def cycle_3():
  # --- Cycle 3 - Circulaire (UI) ---
  movel(apply_correction(p[-0.017788, 0.586142, 0.060004, 3.141576, 0.000000, 0.000000]), a=URSCRIPT_ACCEL*ACCEL_FACTOR, v=0.2500*SPEED_FACTOR)
  sleep(0.2)
  zero_ftsensor()
  sleep(0.2)
  force_mode(MEAS_FRAME, [0, 0, 1, 0, 0, 0], [0, 0, -6.0, 0, 0, 0], 2, [0.008, 0.008, 0.04, 0.35, 0.35, 0.35])
  movel(apply_correction(p[-0.017788, 0.586142, 0.045004, 3.141576, 0.000000, 0.000000]), a=URSCRIPT_ACCEL*ACCEL_FACTOR, v=URSCRIPT_RECONTACT_V*SPEED_FACTOR)
  movel(apply_correction(p[-0.017788, 0.586142, 0.050004, 3.141576, 0.000000, 0.000000]), a=URSCRIPT_ACCEL*ACCEL_FACTOR, v=V_CIRC*SPEED_FACTOR, r=URSCRIPT_BLEND)
  movel(apply_correction(p[-0.011098, 0.583533, 0.050004, 3.141576, 0.000000, 0.000000]), a=URSCRIPT_ACCEL*ACCEL_FACTOR, v=V_CIRC*SPEED_FACTOR, r=URSCRIPT_BLEND)
  movel(apply_correction(p[-0.004916, 0.587048, 0.050004, 3.141576, 0.000000, 0.000000]), a=URSCRIPT_ACCEL*ACCEL_FACTOR, v=V_CIRC*SPEED_FACTOR, r=URSCRIPT_BLEND)
  movel(apply_correction(p[-0.005086, 0.594004, 0.050004, 3.141576, 0.000000, 0.000000]), a=URSCRIPT_ACCEL*ACCEL_FACTOR, v=V_CIRC*SPEED_FACTOR, r=URSCRIPT_BLEND)
  movel(apply_correction(p[-0.011712, 0.596025, 0.050004, 3.141576, 0.000000, 0.000000]), a=URSCRIPT_ACCEL*ACCEL_FACTOR, v=V_CIRC*SPEED_FACTOR, r=URSCRIPT_BLEND)
  movel(apply_correction(p[-0.016472, 0.590781, 0.050004, 3.141576, 0.000000, 0.000000]), a=URSCRIPT_ACCEL*ACCEL_FACTOR, v=V_CIRC*SPEED_FACTOR, r=URSCRIPT_BLEND)
  movel(apply_correction(p[-0.015164, 0.583730, 0.050004, 3.141576, 0.000000, 0.000000]), a=URSCRIPT_ACCEL*ACCEL_FACTOR, v=V_CIRC*SPEED_FACTOR, r=URSCRIPT_BLEND)
  movel(apply_correction(p[-0.009065, 0.579930, 0.050004, 3.141576, 0.000000, 0.000000]), a=URSCRIPT_ACCEL*ACCEL_FACTOR, v=V_CIRC*SPEED_FACTOR, r=URSCRIPT_BLEND)
  movel(apply_correction(p[-0.002264, 0.582086, 0.050004, 3.141576, 0.000000, 0.000000]), a=URSCRIPT_ACCEL*ACCEL_FACTOR, v=V_CIRC*SPEED_FACTOR, r=URSCRIPT_BLEND)
  movel(apply_correction(p[-0.000623, 0.588885, 0.050004, 3.141576, 0.000000, 0.000000]), a=URSCRIPT_ACCEL*ACCEL_FACTOR, v=V_CIRC*SPEED_FACTOR, r=URSCRIPT_BLEND)
  movel(apply_correction(p[-0.006418, 0.592643, 0.050004, 3.141576, 0.000000, 0.000000]), a=URSCRIPT_ACCEL*ACCEL_FACTOR, v=V_CIRC*SPEED_FACTOR, r=URSCRIPT_BLEND)
  movel(apply_correction(p[-0.012226, 0.588648, 0.050004, 3.141576, 0.000000, 0.000000]), a=URSCRIPT_ACCEL*ACCEL_FACTOR, v=V_CIRC*SPEED_FACTOR, r=URSCRIPT_BLEND)
  movel(apply_correction(p[-0.012291, 0.581489, 0.050004, 3.141576, 0.000000, 0.000000]), a=URSCRIPT_ACCEL*ACCEL_FACTOR, v=V_CIRC*SPEED_FACTOR, r=URSCRIPT_BLEND)
  movel(apply_correction(p[-0.006988, 0.576638, 0.050004, 3.141576, 0.000000, 0.000000]), a=URSCRIPT_ACCEL*ACCEL_FACTOR, v=V_CIRC*SPEED_FACTOR, r=URSCRIPT_BLEND)
  movel(apply_correction(p[0.000125, 0.577386, 0.050004, 3.141576, 0.000000, 0.000000]), a=URSCRIPT_ACCEL*ACCEL_FACTOR, v=V_CIRC*SPEED_FACTOR, r=URSCRIPT_BLEND)
  movel(apply_correction(p[0.003408, 0.583603, 0.050004, 3.141576, 0.000000, 0.000000]), a=URSCRIPT_ACCEL*ACCEL_FACTOR, v=V_CIRC*SPEED_FACTOR, r=URSCRIPT_BLEND)
  movel(apply_correction(p[-0.001104, 0.588825, 0.050004, 3.141576, 0.000000, 0.000000]), a=URSCRIPT_ACCEL*ACCEL_FACTOR, v=V_CIRC*SPEED_FACTOR, r=URSCRIPT_BLEND)
  movel(apply_correction(p[-0.007670, 0.586361, 0.050004, 3.141576, 0.000000, 0.000000]), a=URSCRIPT_ACCEL*ACCEL_FACTOR, v=V_CIRC*SPEED_FACTOR, r=URSCRIPT_BLEND)
  movel(apply_correction(p[-0.009144, 0.579371, 0.050004, 3.141576, 0.000000, 0.000000]), a=URSCRIPT_ACCEL*ACCEL_FACTOR, v=V_CIRC*SPEED_FACTOR, r=URSCRIPT_BLEND)
  movel(apply_correction(p[-0.004813, 0.573634, 0.050004, 3.141576, 0.000000, 0.000000]), a=URSCRIPT_ACCEL*ACCEL_FACTOR, v=V_CIRC*SPEED_FACTOR, r=URSCRIPT_BLEND)
  movel(apply_correction(p[0.002324, 0.572985, 0.050004, 3.141576, 0.000000, 0.000000]), a=URSCRIPT_ACCEL*ACCEL_FACTOR, v=V_CIRC*SPEED_FACTOR, r=URSCRIPT_BLEND)
  movel(apply_correction(p[0.006999, 0.578286, 0.050004, 3.141576, 0.000000, 0.000000]), a=URSCRIPT_ACCEL*ACCEL_FACTOR, v=V_CIRC*SPEED_FACTOR, r=URSCRIPT_BLEND)
  movel(apply_correction(p[0.004110, 0.584567, 0.050004, 3.141576, 0.000000, 0.000000]), a=URSCRIPT_ACCEL*ACCEL_FACTOR, v=V_CIRC*SPEED_FACTOR, r=URSCRIPT_BLEND)
  movel(apply_correction(p[-0.002829, 0.583846, 0.050004, 3.141576, 0.000000, 0.000000]), a=URSCRIPT_ACCEL*ACCEL_FACTOR, v=V_CIRC*SPEED_FACTOR, r=URSCRIPT_BLEND)
  movel(apply_correction(p[-0.005691, 0.577324, 0.050004, 3.141576, 0.000000, 0.000000]), a=URSCRIPT_ACCEL*ACCEL_FACTOR, v=V_CIRC*SPEED_FACTOR, r=URSCRIPT_BLEND)
  movel(apply_correction(p[-0.002490, 0.570894, 0.050004, 3.141576, 0.000000, 0.000000]), a=URSCRIPT_ACCEL*ACCEL_FACTOR, v=V_CIRC*SPEED_FACTOR, r=URSCRIPT_BLEND)
  movel(apply_correction(p[0.004406, 0.568905, 0.050004, 3.141576, 0.000000, 0.000000]), a=URSCRIPT_ACCEL*ACCEL_FACTOR, v=V_CIRC*SPEED_FACTOR, r=URSCRIPT_BLEND)
  movel(apply_correction(p[0.010171, 0.573044, 0.050004, 3.141576, 0.000000, 0.000000]), a=URSCRIPT_ACCEL*ACCEL_FACTOR, v=V_CIRC*SPEED_FACTOR, r=URSCRIPT_BLEND)
  movel(apply_correction(p[0.009098, 0.579900, 0.050004, 3.141576, 0.000000, 0.000000]), a=URSCRIPT_ACCEL*ACCEL_FACTOR, v=V_CIRC*SPEED_FACTOR, r=URSCRIPT_BLEND)
  movel(apply_correction(p[0.002251, 0.581029, 0.050004, 3.141576, 0.000000, 0.000000]), a=URSCRIPT_ACCEL*ACCEL_FACTOR, v=V_CIRC*SPEED_FACTOR, r=URSCRIPT_BLEND)
  movel(apply_correction(p[-0.001925, 0.575290, 0.050004, 3.141576, 0.000000, 0.000000]), a=URSCRIPT_ACCEL*ACCEL_FACTOR, v=V_CIRC*SPEED_FACTOR, r=URSCRIPT_BLEND)
  movel(apply_correction(p[0.000027, 0.568386, 0.050004, 3.141576, 0.000000, 0.000000]), a=URSCRIPT_ACCEL*ACCEL_FACTOR, v=V_CIRC*SPEED_FACTOR, r=URSCRIPT_BLEND)
  movel(apply_correction(p[0.006439, 0.565146, 0.050005, 3.141576, 0.000000, 0.000000]), a=URSCRIPT_ACCEL*ACCEL_FACTOR, v=V_CIRC*SPEED_FACTOR, r=URSCRIPT_BLEND)
  movel(apply_correction(p[0.012978, 0.567972, 0.050004, 3.141576, 0.000000, 0.000000]), a=URSCRIPT_ACCEL*ACCEL_FACTOR, v=V_CIRC*SPEED_FACTOR, r=URSCRIPT_BLEND)
  movel(apply_correction(p[0.013753, 0.574903, 0.050004, 3.141576, 0.000000, 0.000000]), a=URSCRIPT_ACCEL*ACCEL_FACTOR, v=V_CIRC*SPEED_FACTOR, r=URSCRIPT_BLEND)
  movel(apply_correction(p[0.007496, 0.577845, 0.050004, 3.141576, 0.000000, 0.000000]), a=URSCRIPT_ACCEL*ACCEL_FACTOR, v=V_CIRC*SPEED_FACTOR, r=URSCRIPT_BLEND)
  movel(apply_correction(p[0.002166, 0.573206, 0.050004, 3.141576, 0.000000, 0.000000]), a=URSCRIPT_ACCEL*ACCEL_FACTOR, v=V_CIRC*SPEED_FACTOR, r=URSCRIPT_BLEND)
  movel(apply_correction(p[0.002775, 0.566066, 0.050004, 3.141576, 0.000000, 0.000000]), a=URSCRIPT_ACCEL*ACCEL_FACTOR, v=V_CIRC*SPEED_FACTOR, r=URSCRIPT_BLEND)
  movel(apply_correction(p[0.008487, 0.561706, 0.050005, 3.141576, 0.000000, 0.000000]), a=URSCRIPT_ACCEL*ACCEL_FACTOR, v=V_CIRC*SPEED_FACTOR, r=URSCRIPT_BLEND)
  movel(apply_correction(p[0.015475, 0.563167, 0.050005, 3.141576, 0.000000, 0.000000]), a=URSCRIPT_ACCEL*ACCEL_FACTOR, v=V_CIRC*SPEED_FACTOR, r=URSCRIPT_BLEND)
  movel(apply_correction(p[0.017743, 0.569730, 0.050004, 3.141576, 0.000000, 0.000000]), a=URSCRIPT_ACCEL*ACCEL_FACTOR, v=V_CIRC*SPEED_FACTOR, r=URSCRIPT_BLEND)
  movel(apply_correction(p[0.012260, 0.573881, 0.050004, 3.141576, 0.000000, 0.000000]), a=URSCRIPT_ACCEL*ACCEL_FACTOR, v=V_CIRC*SPEED_FACTOR, r=URSCRIPT_BLEND)
  movel(apply_correction(p[0.005935, 0.570677, 0.050004, 3.141576, 0.000000, 0.000000]), a=URSCRIPT_ACCEL*ACCEL_FACTOR, v=V_CIRC*SPEED_FACTOR, r=URSCRIPT_BLEND)
  movel(apply_correction(p[0.004428, 0.563644, 0.050005, 3.141576, 0.000000, 0.000000]), a=URSCRIPT_ACCEL*ACCEL_FACTOR, v=V_CIRC*SPEED_FACTOR, r=URSCRIPT_BLEND)
  movel(apply_correction(p[0.008552, 0.557768, 0.050005, 3.141576, 0.000000, 0.000000]), a=URSCRIPT_ACCEL*ACCEL_FACTOR, v=V_CIRC*SPEED_FACTOR, r=URSCRIPT_BLEND)
  movel(apply_correction(p[0.015598, 0.557554, 0.050005, 3.141576, 0.000000, 0.000000]), a=URSCRIPT_ACCEL*ACCEL_FACTOR, v=V_CIRC*SPEED_FACTOR, r=URSCRIPT_BLEND)
  movel(apply_correction(p[0.018398, 0.563819, 0.050005, 3.141576, 0.000000, 0.000000]), a=URSCRIPT_ACCEL*ACCEL_FACTOR, v=V_CIRC*SPEED_FACTOR, r=URSCRIPT_BLEND)
  movel(apply_correction(p[0.013349, 0.568656, 0.050004, 3.141576, 0.000000, 0.000000]), a=URSCRIPT_ACCEL*ACCEL_FACTOR, v=V_CIRC*SPEED_FACTOR, r=URSCRIPT_BLEND)
  movel(apply_correction(p[0.006365, 0.567164, 0.050004, 3.141576, 0.000000, 0.000000]), a=URSCRIPT_ACCEL*ACCEL_FACTOR, v=V_CIRC*SPEED_FACTOR, r=URSCRIPT_BLEND)
  movel(apply_correction(p[0.002726, 0.560986, 0.050005, 3.141576, 0.000000, 0.000000]), a=URSCRIPT_ACCEL*ACCEL_FACTOR, v=V_CIRC*SPEED_FACTOR, r=URSCRIPT_BLEND)
  movel(apply_correction(p[0.004975, 0.554229, 0.050005, 3.141576, 0.000000, 0.000000]), a=URSCRIPT_ACCEL*ACCEL_FACTOR, v=V_CIRC*SPEED_FACTOR, r=URSCRIPT_BLEND)
  movel(apply_correction(p[0.011813, 0.552992, 0.050005, 3.141576, 0.000000, 0.000000]), a=URSCRIPT_ACCEL*ACCEL_FACTOR, v=V_CIRC*SPEED_FACTOR, r=URSCRIPT_BLEND)
  movel(apply_correction(p[0.015059, 0.559096, 0.050005, 3.141576, 0.000000, 0.000000]), a=URSCRIPT_ACCEL*ACCEL_FACTOR, v=V_CIRC*SPEED_FACTOR, r=URSCRIPT_BLEND)
  movel(apply_correction(p[0.011046, 0.564958, 0.050005, 3.141576, 0.000000, 0.000000]), a=URSCRIPT_ACCEL*ACCEL_FACTOR, v=V_CIRC*SPEED_FACTOR, r=URSCRIPT_BLEND)
  movel(apply_correction(p[0.003896, 0.565651, 0.050004, 3.141576, 0.000000, 0.000000]), a=URSCRIPT_ACCEL*ACCEL_FACTOR, v=V_CIRC*SPEED_FACTOR, r=URSCRIPT_BLEND)
  movel(apply_correction(p[-0.001449, 0.560893, 0.050005, 3.141576, 0.000000, 0.000000]), a=URSCRIPT_ACCEL*ACCEL_FACTOR, v=V_CIRC*SPEED_FACTOR, r=URSCRIPT_BLEND)
  movel(apply_correction(p[-0.000730, 0.553895, 0.050005, 3.141576, 0.000000, 0.000000]), a=URSCRIPT_ACCEL*ACCEL_FACTOR, v=V_CIRC*SPEED_FACTOR, r=URSCRIPT_BLEND)
  movel(apply_correction(p[0.005938, 0.552136, 0.050005, 3.141576, 0.000000, 0.000000]), a=URSCRIPT_ACCEL*ACCEL_FACTOR, v=V_CIRC*SPEED_FACTOR, r=URSCRIPT_BLEND)
  movel(apply_correction(p[0.010014, 0.557869, 0.050005, 3.141576, 0.000000, 0.000000]), a=URSCRIPT_ACCEL*ACCEL_FACTOR, v=V_CIRC*SPEED_FACTOR, r=URSCRIPT_BLEND)
  movel(apply_correction(p[0.007718, 0.564641, 0.050005, 3.141576, 0.000000, 0.000000]), a=URSCRIPT_ACCEL*ACCEL_FACTOR, v=V_CIRC*SPEED_FACTOR, r=URSCRIPT_BLEND)
  movel(apply_correction(p[0.001166, 0.567570, 0.050004, 3.141576, 0.000000, 0.000000]), a=URSCRIPT_ACCEL*ACCEL_FACTOR, v=V_CIRC*SPEED_FACTOR, r=URSCRIPT_BLEND)
  movel(apply_correction(p[-0.005246, 0.564498, 0.050005, 3.141576, 0.000000, 0.000000]), a=URSCRIPT_ACCEL*ACCEL_FACTOR, v=V_CIRC*SPEED_FACTOR, r=URSCRIPT_BLEND)
  movel(apply_correction(p[-0.005654, 0.557540, 0.050005, 3.141576, 0.000000, 0.000000]), a=URSCRIPT_ACCEL*ACCEL_FACTOR, v=V_CIRC*SPEED_FACTOR, r=URSCRIPT_BLEND)
  movel(apply_correction(p[0.000763, 0.554955, 0.050005, 3.141576, 0.000000, 0.000000]), a=URSCRIPT_ACCEL*ACCEL_FACTOR, v=V_CIRC*SPEED_FACTOR, r=URSCRIPT_BLEND)
  movel(apply_correction(p[0.005879, 0.559839, 0.050005, 3.141576, 0.000000, 0.000000]), a=URSCRIPT_ACCEL*ACCEL_FACTOR, v=V_CIRC*SPEED_FACTOR, r=URSCRIPT_BLEND)
  movel(apply_correction(p[0.004993, 0.566952, 0.050004, 3.141576, 0.000000, 0.000000]), a=URSCRIPT_ACCEL*ACCEL_FACTOR, v=V_CIRC*SPEED_FACTOR, r=URSCRIPT_BLEND)
  movel(apply_correction(p[-0.000876, 0.571099, 0.050004, 3.141576, 0.000000, 0.000000]), a=URSCRIPT_ACCEL*ACCEL_FACTOR, v=V_CIRC*SPEED_FACTOR, r=URSCRIPT_BLEND)
  movel(apply_correction(p[-0.007807, 0.569384, 0.050004, 3.141576, 0.000000, 0.000000]), a=URSCRIPT_ACCEL*ACCEL_FACTOR, v=V_CIRC*SPEED_FACTOR, r=URSCRIPT_BLEND)
  movel(apply_correction(p[-0.009985, 0.562724, 0.050005, 3.141576, 0.000000, 0.000000]), a=URSCRIPT_ACCEL*ACCEL_FACTOR, v=V_CIRC*SPEED_FACTOR, r=URSCRIPT_BLEND)
  movel(apply_correction(p[-0.004550, 0.558471, 0.050005, 3.141576, 0.000000, 0.000000]), a=URSCRIPT_ACCEL*ACCEL_FACTOR, v=V_CIRC*SPEED_FACTOR, r=URSCRIPT_BLEND)
  movel(apply_correction(p[0.001532, 0.562013, 0.050005, 3.141576, 0.000000, 0.000000]), a=URSCRIPT_ACCEL*ACCEL_FACTOR, v=V_CIRC*SPEED_FACTOR, r=URSCRIPT_BLEND)
  movel(apply_correction(p[0.002038, 0.569150, 0.050004, 3.141576, 0.000000, 0.000000]), a=URSCRIPT_ACCEL*ACCEL_FACTOR, v=V_CIRC*SPEED_FACTOR, r=URSCRIPT_BLEND)
  movel(apply_correction(p[-0.002979, 0.574298, 0.050004, 3.141576, 0.000000, 0.000000]), a=URSCRIPT_ACCEL*ACCEL_FACTOR, v=V_CIRC*SPEED_FACTOR, r=URSCRIPT_BLEND)
  movel(apply_correction(p[-0.010128, 0.573991, 0.050004, 3.141576, 0.000000, 0.000000]), a=URSCRIPT_ACCEL*ACCEL_FACTOR, v=V_CIRC*SPEED_FACTOR, r=URSCRIPT_BLEND)
  movel(apply_correction(p[-0.013879, 0.568031, 0.050004, 3.141576, 0.000000, 0.000000]), a=URSCRIPT_ACCEL*ACCEL_FACTOR, v=V_CIRC*SPEED_FACTOR, r=URSCRIPT_BLEND)
  movel(apply_correction(p[-0.009845, 0.562427, 0.050005, 3.141576, 0.000000, 0.000000]), a=URSCRIPT_ACCEL*ACCEL_FACTOR, v=V_CIRC*SPEED_FACTOR, r=URSCRIPT_BLEND)
  movel(apply_correction(p[-0.003119, 0.564364, 0.050005, 3.141576, 0.000000, 0.000000]), a=URSCRIPT_ACCEL*ACCEL_FACTOR, v=V_CIRC*SPEED_FACTOR, r=URSCRIPT_BLEND)
  movel(apply_correction(p[-0.001202, 0.571240, 0.050004, 3.141576, 0.000000, 0.000000]), a=URSCRIPT_ACCEL*ACCEL_FACTOR, v=V_CIRC*SPEED_FACTOR, r=URSCRIPT_BLEND)
  movel(apply_correction(p[-0.005195, 0.577216, 0.050004, 3.141576, 0.000000, 0.000000]), a=URSCRIPT_ACCEL*ACCEL_FACTOR, v=V_CIRC*SPEED_FACTOR, r=URSCRIPT_BLEND)
  movel(apply_correction(p[-0.012283, 0.578294, 0.050004, 3.141576, 0.000000, 0.000000]), a=URSCRIPT_ACCEL*ACCEL_FACTOR, v=V_CIRC*SPEED_FACTOR, r=URSCRIPT_BLEND)
  movel(apply_correction(p[-0.017334, 0.573336, 0.050004, 3.141576, 0.000000, 0.000000]), a=URSCRIPT_ACCEL*ACCEL_FACTOR, v=V_CIRC*SPEED_FACTOR, r=URSCRIPT_BLEND)
  movel(apply_correction(p[-0.015002, 0.566819, 0.050004, 3.141576, 0.000000, 0.000000]), a=URSCRIPT_ACCEL*ACCEL_FACTOR, v=V_CIRC*SPEED_FACTOR, r=URSCRIPT_BLEND)
  movel(apply_correction(p[-0.008039, 0.566966, 0.050004, 3.141576, 0.000000, 0.000000]), a=URSCRIPT_ACCEL*ACCEL_FACTOR, v=V_CIRC*SPEED_FACTOR, r=URSCRIPT_BLEND)
  movel(apply_correction(p[-0.004752, 0.573277, 0.050004, 3.141576, 0.000000, 0.000000]), a=URSCRIPT_ACCEL*ACCEL_FACTOR, v=V_CIRC*SPEED_FACTOR, r=URSCRIPT_BLEND)
  movel(apply_correction(p[-0.007574, 0.579880, 0.050004, 3.141576, 0.000000, 0.000000]), a=URSCRIPT_ACCEL*ACCEL_FACTOR, v=V_CIRC*SPEED_FACTOR, r=URSCRIPT_BLEND)
  movel(apply_correction(p[-0.014343, 0.582272, 0.050004, 3.141576, 0.000000, 0.000000]), a=URSCRIPT_ACCEL*ACCEL_FACTOR, v=V_CIRC*SPEED_FACTOR, r=URSCRIPT_BLEND)
  movel(apply_correction(p[-0.020386, 0.578533, 0.050004, 3.141576, 0.000000, 0.000000]), a=URSCRIPT_ACCEL*ACCEL_FACTOR, v=V_CIRC*SPEED_FACTOR, r=URSCRIPT_BLEND)
  movel(apply_correction(p[-0.019895, 0.571600, 0.050004, 3.141576, 0.000000, 0.000000]), a=URSCRIPT_ACCEL*ACCEL_FACTOR, v=V_CIRC*SPEED_FACTOR, r=URSCRIPT_BLEND)
  movel(apply_correction(p[-0.013179, 0.569890, 0.050004, 3.141576, 0.000000, 0.000000]), a=URSCRIPT_ACCEL*ACCEL_FACTOR, v=V_CIRC*SPEED_FACTOR, r=URSCRIPT_BLEND)
  movel(apply_correction(p[-0.008631, 0.575334, 0.050004, 3.141576, 0.000000, 0.000000]), a=URSCRIPT_ACCEL*ACCEL_FACTOR, v=V_CIRC*SPEED_FACTOR, r=URSCRIPT_BLEND)
  movel(apply_correction(p[-0.010345, 0.582287, 0.050004, 3.141576, 0.000000, 0.000000]), a=URSCRIPT_ACCEL*ACCEL_FACTOR, v=V_CIRC*SPEED_FACTOR, r=URSCRIPT_BLEND)
  movel(apply_correction(p[-0.016696, 0.585620, 0.050004, 3.141576, 0.000000, 0.000000]), a=URSCRIPT_ACCEL*ACCEL_FACTOR, v=V_CIRC*SPEED_FACTOR, r=URSCRIPT_BLEND)
  movel(apply_correction(p[-0.023362, 0.583056, 0.050004, 3.141576, 0.000000, 0.000000]), a=URSCRIPT_ACCEL*ACCEL_FACTOR, v=V_CIRC*SPEED_FACTOR, r=URSCRIPT_BLEND)
  movel(apply_correction(p[-0.025236, 0.576243, 0.050004, 3.141576, 0.000000, 0.000000]), a=URSCRIPT_ACCEL*ACCEL_FACTOR, v=V_CIRC*SPEED_FACTOR, r=URSCRIPT_BLEND)
  movel(apply_correction(p[-0.020034, 0.571653, 0.050004, 3.141576, 0.000000, 0.000000]), a=URSCRIPT_ACCEL*ACCEL_FACTOR, v=V_CIRC*SPEED_FACTOR, r=URSCRIPT_BLEND)
  movel(apply_correction(p[-0.014038, 0.575090, 0.050004, 3.141576, 0.000000, 0.000000]), a=URSCRIPT_ACCEL*ACCEL_FACTOR, v=V_CIRC*SPEED_FACTOR, r=URSCRIPT_BLEND)
  movel(apply_correction(p[-0.014738, 0.582089, 0.050004, 3.141576, 0.000000, 0.000000]), a=URSCRIPT_ACCEL*ACCEL_FACTOR, v=V_CIRC*SPEED_FACTOR, r=URSCRIPT_BLEND)
  movel(apply_correction(p[-0.020976, 0.585534, 0.050004, 3.141576, 0.000000, 0.000000]), a=URSCRIPT_ACCEL*ACCEL_FACTOR, v=V_CIRC*SPEED_FACTOR, r=URSCRIPT_BLEND)
  movel(apply_correction(p[-0.027687, 0.583050, 0.050004, 3.141576, 0.000000, 0.000000]), a=URSCRIPT_ACCEL*ACCEL_FACTOR, v=V_CIRC*SPEED_FACTOR, r=URSCRIPT_BLEND)
  movel(apply_correction(p[-0.030305, 0.576399, 0.050004, 3.141576, 0.000000, 0.000000]), a=URSCRIPT_ACCEL*ACCEL_FACTOR, v=V_CIRC*SPEED_FACTOR, r=URSCRIPT_BLEND)
  movel(apply_correction(p[-0.026697, 0.570296, 0.050004, 3.141576, 0.000000, 0.000000]), a=URSCRIPT_ACCEL*ACCEL_FACTOR, v=V_CIRC*SPEED_FACTOR, r=URSCRIPT_BLEND)
  movel(apply_correction(p[-0.019718, 0.570534, 0.050004, 3.141576, 0.000000, 0.000000]), a=URSCRIPT_ACCEL*ACCEL_FACTOR, v=V_CIRC*SPEED_FACTOR, r=URSCRIPT_BLEND)
  movel(apply_correction(p[-0.017643, 0.577142, 0.050004, 3.141576, 0.000000, 0.000000]), a=URSCRIPT_ACCEL*ACCEL_FACTOR, v=V_CIRC*SPEED_FACTOR, r=URSCRIPT_BLEND)
  movel(apply_correction(p[-0.023092, 0.581572, 0.050004, 3.141576, 0.000000, 0.000000]), a=URSCRIPT_ACCEL*ACCEL_FACTOR, v=V_CIRC*SPEED_FACTOR, r=URSCRIPT_BLEND)
  movel(apply_correction(p[-0.029871, 0.579381, 0.050004, 3.141576, 0.000000, 0.000000]), a=URSCRIPT_ACCEL*ACCEL_FACTOR, v=V_CIRC*SPEED_FACTOR, r=URSCRIPT_BLEND)
  movel(apply_correction(p[-0.032536, 0.572708, 0.050004, 3.141576, 0.000000, 0.000000]), a=URSCRIPT_ACCEL*ACCEL_FACTOR, v=V_CIRC*SPEED_FACTOR, r=URSCRIPT_BLEND)
  movel(apply_correction(p[-0.029339, 0.566277, 0.050004, 3.141576, 0.000000, 0.000000]), a=URSCRIPT_ACCEL*ACCEL_FACTOR, v=V_CIRC*SPEED_FACTOR, r=URSCRIPT_BLEND)
  movel(apply_correction(p[-0.022399, 0.564726, 0.050005, 3.141576, 0.000000, 0.000000]), a=URSCRIPT_ACCEL*ACCEL_FACTOR, v=V_CIRC*SPEED_FACTOR, r=URSCRIPT_BLEND)
  movel(apply_correction(p[-0.017535, 0.569747, 0.050004, 3.141576, 0.000000, 0.000000]), a=URSCRIPT_ACCEL*ACCEL_FACTOR, v=V_CIRC*SPEED_FACTOR, r=URSCRIPT_BLEND)
  movel(apply_correction(p[-0.020477, 0.575989, 0.050004, 3.141576, 0.000000, 0.000000]), a=URSCRIPT_ACCEL*ACCEL_FACTOR, v=V_CIRC*SPEED_FACTOR, r=URSCRIPT_BLEND)
  movel(apply_correction(p[-0.027450, 0.575397, 0.050004, 3.141576, 0.000000, 0.000000]), a=URSCRIPT_ACCEL*ACCEL_FACTOR, v=V_CIRC*SPEED_FACTOR, r=URSCRIPT_BLEND)
  movel(apply_correction(p[-0.030496, 0.568956, 0.050004, 3.141576, 0.000000, 0.000000]), a=URSCRIPT_ACCEL*ACCEL_FACTOR, v=V_CIRC*SPEED_FACTOR, r=URSCRIPT_BLEND)
  movel(apply_correction(p[-0.027445, 0.562453, 0.050005, 3.141576, 0.000000, 0.000000]), a=URSCRIPT_ACCEL*ACCEL_FACTOR, v=V_CIRC*SPEED_FACTOR, r=URSCRIPT_BLEND)
  movel(apply_correction(p[-0.020600, 0.560297, 0.050005, 3.141576, 0.000000, 0.000000]), a=URSCRIPT_ACCEL*ACCEL_FACTOR, v=V_CIRC*SPEED_FACTOR, r=URSCRIPT_BLEND)
  movel(apply_correction(p[-0.014717, 0.564274, 0.050005, 3.141576, 0.000000, 0.000000]), a=URSCRIPT_ACCEL*ACCEL_FACTOR, v=V_CIRC*SPEED_FACTOR, r=URSCRIPT_BLEND)
  movel(apply_correction(p[-0.015552, 0.571170, 0.050004, 3.141576, 0.000000, 0.000000]), a=URSCRIPT_ACCEL*ACCEL_FACTOR, v=V_CIRC*SPEED_FACTOR, r=URSCRIPT_BLEND)
  movel(apply_correction(p[-0.022352, 0.572534, 0.050004, 3.141576, 0.000000, 0.000000]), a=URSCRIPT_ACCEL*ACCEL_FACTOR, v=V_CIRC*SPEED_FACTOR, r=URSCRIPT_BLEND)
  movel(apply_correction(p[-0.026686, 0.566919, 0.050004, 3.141576, 0.000000, 0.000000]), a=URSCRIPT_ACCEL*ACCEL_FACTOR, v=V_CIRC*SPEED_FACTOR, r=URSCRIPT_BLEND)
  movel(apply_correction(p[-0.024903, 0.559969, 0.050005, 3.141576, 0.000000, 0.000000]), a=URSCRIPT_ACCEL*ACCEL_FACTOR, v=V_CIRC*SPEED_FACTOR, r=URSCRIPT_BLEND)
  movel(apply_correction(p[-0.018568, 0.556581, 0.050005, 3.141576, 0.000000, 0.000000]), a=URSCRIPT_ACCEL*ACCEL_FACTOR, v=V_CIRC*SPEED_FACTOR, r=URSCRIPT_BLEND)
  movel(apply_correction(p[-0.011952, 0.559230, 0.050005, 3.141576, 0.000000, 0.000000]), a=URSCRIPT_ACCEL*ACCEL_FACTOR, v=V_CIRC*SPEED_FACTOR, r=URSCRIPT_BLEND)
  movel(apply_correction(p[-0.010947, 0.566137, 0.050004, 3.141576, 0.000000, 0.000000]), a=URSCRIPT_ACCEL*ACCEL_FACTOR, v=V_CIRC*SPEED_FACTOR, r=URSCRIPT_BLEND)
  movel(apply_correction(p[-0.017092, 0.569298, 0.050004, 3.141576, 0.000000, 0.000000]), a=URSCRIPT_ACCEL*ACCEL_FACTOR, v=V_CIRC*SPEED_FACTOR, r=URSCRIPT_BLEND)
  movel(apply_correction(p[-0.022556, 0.564825, 0.050005, 3.141576, 0.000000, 0.000000]), a=URSCRIPT_ACCEL*ACCEL_FACTOR, v=V_CIRC*SPEED_FACTOR, r=URSCRIPT_BLEND)
  movel(apply_correction(p[-0.022123, 0.557672, 0.050005, 3.141576, 0.000000, 0.000000]), a=URSCRIPT_ACCEL*ACCEL_FACTOR, v=V_CIRC*SPEED_FACTOR, r=URSCRIPT_BLEND)
  movel(apply_correction(p[-0.016514, 0.553178, 0.050005, 3.141576, 0.000000, 0.000000]), a=URSCRIPT_ACCEL*ACCEL_FACTOR, v=V_CIRC*SPEED_FACTOR, r=URSCRIPT_BLEND)
  movel(apply_correction(p[-0.009477, 0.554429, 0.050005, 3.141576, 0.000000, 0.000000]), a=URSCRIPT_ACCEL*ACCEL_FACTOR, v=V_CIRC*SPEED_FACTOR, r=URSCRIPT_BLEND)
  movel(apply_correction(p[-0.006757, 0.560900, 0.050005, 3.141576, 0.000000, 0.000000]), a=URSCRIPT_ACCEL*ACCEL_FACTOR, v=V_CIRC*SPEED_FACTOR, r=URSCRIPT_BLEND)
  movel(apply_correction(p[-0.011771, 0.565641, 0.050004, 3.141576, 0.000000, 0.000000]), a=URSCRIPT_ACCEL*ACCEL_FACTOR, v=V_CIRC*SPEED_FACTOR, r=URSCRIPT_BLEND)
  movel(apply_correction(p[-0.018106, 0.562599, 0.050005, 3.141576, 0.000000, 0.000000]), a=URSCRIPT_ACCEL*ACCEL_FACTOR, v=V_CIRC*SPEED_FACTOR, r=URSCRIPT_BLEND)
  movel(apply_correction(p[-0.019075, 0.555515, 0.050005, 3.141576, 0.000000, 0.000000]), a=URSCRIPT_ACCEL*ACCEL_FACTOR, v=V_CIRC*SPEED_FACTOR, r=URSCRIPT_BLEND)
  movel(apply_correction(p[-0.014379, 0.550076, 0.050005, 3.141576, 0.000000, 0.000000]), a=URSCRIPT_ACCEL*ACCEL_FACTOR, v=V_CIRC*SPEED_FACTOR, r=URSCRIPT_BLEND)
  movel(apply_correction(p[-0.007220, 0.549921, 0.050005, 3.141576, 0.000000, 0.000000]), a=URSCRIPT_ACCEL*ACCEL_FACTOR, v=V_CIRC*SPEED_FACTOR, r=URSCRIPT_BLEND)
  movel(apply_correction(p[-0.003008, 0.555581, 0.050005, 3.141576, 0.000000, 0.000000]), a=URSCRIPT_ACCEL*ACCEL_FACTOR, v=V_CIRC*SPEED_FACTOR, r=URSCRIPT_BLEND)
  movel(apply_correction(p[-0.006508, 0.561538, 0.050005, 3.141576, 0.000000, 0.000000]), a=URSCRIPT_ACCEL*ACCEL_FACTOR, v=V_CIRC*SPEED_FACTOR, r=URSCRIPT_BLEND)
  movel(apply_correction(p[-0.013362, 0.560174, 0.050005, 3.141576, 0.000000, 0.000000]), a=URSCRIPT_ACCEL*ACCEL_FACTOR, v=V_CIRC*SPEED_FACTOR, r=URSCRIPT_BLEND)
  movel(apply_correction(p[-0.015736, 0.553449, 0.050005, 3.141576, 0.000000, 0.000000]), a=URSCRIPT_ACCEL*ACCEL_FACTOR, v=V_CIRC*SPEED_FACTOR, r=URSCRIPT_BLEND)
  movel(apply_correction(p[-0.012114, 0.547244, 0.050005, 3.141576, 0.000000, 0.000000]), a=URSCRIPT_ACCEL*ACCEL_FACTOR, v=V_CIRC*SPEED_FACTOR, r=URSCRIPT_BLEND)
  movel(apply_correction(p[-0.005103, 0.545724, 0.050005, 3.141576, 0.000000, 0.000000]), a=URSCRIPT_ACCEL*ACCEL_FACTOR, v=V_CIRC*SPEED_FACTOR, r=URSCRIPT_BLEND)
  movel(apply_correction(p[0.000267, 0.550317, 0.050005, 3.141576, 0.000000, 0.000000]), a=URSCRIPT_ACCEL*ACCEL_FACTOR, v=V_CIRC*SPEED_FACTOR, r=URSCRIPT_BLEND)
  movel(apply_correction(p[-0.001550, 0.556944, 0.050005, 3.141576, 0.000000, 0.000000]), a=URSCRIPT_ACCEL*ACCEL_FACTOR, v=V_CIRC*SPEED_FACTOR, r=URSCRIPT_BLEND)
  movel(apply_correction(p[-0.008498, 0.557307, 0.050005, 3.141576, 0.000000, 0.000000]), a=URSCRIPT_ACCEL*ACCEL_FACTOR, v=V_CIRC*SPEED_FACTOR, r=URSCRIPT_BLEND)
  movel(apply_correction(p[-0.012498, 0.551407, 0.050005, 3.141576, 0.000000, 0.000000]), a=URSCRIPT_ACCEL*ACCEL_FACTOR, v=V_CIRC*SPEED_FACTOR, r=URSCRIPT_BLEND)
  movel(apply_correction(p[-0.010765, 0.544449, 0.050005, 3.141576, 0.000000, 0.000000]), a=URSCRIPT_ACCEL*ACCEL_FACTOR, v=V_CIRC*SPEED_FACTOR, r=URSCRIPT_BLEND)
  movel(apply_correction(p[-0.004471, 0.541100, 0.050005, 3.141576, 0.000000, 0.000000]), a=URSCRIPT_ACCEL*ACCEL_FACTOR, v=V_CIRC*SPEED_FACTOR, r=URSCRIPT_BLEND)
  movel(apply_correction(p[0.001548, 0.544594, 0.050005, 3.141576, 0.000000, 0.000000]), a=URSCRIPT_ACCEL*ACCEL_FACTOR, v=V_CIRC*SPEED_FACTOR, r=URSCRIPT_BLEND)
  movel(apply_correction(p[0.000165, 0.551320, 0.050005, 3.141576, 0.000000, 0.000000]), a=URSCRIPT_ACCEL*ACCEL_FACTOR, v=V_CIRC*SPEED_FACTOR, r=URSCRIPT_BLEND)
  movel(apply_correction(p[-0.006728, 0.552924, 0.050005, 3.141576, 0.000000, 0.000000]), a=URSCRIPT_ACCEL*ACCEL_FACTOR, v=V_CIRC*SPEED_FACTOR, r=URSCRIPT_BLEND)
  movel(apply_correction(p[-0.012333, 0.548421, 0.050005, 3.141576, 0.000000, 0.000000]), a=URSCRIPT_ACCEL*ACCEL_FACTOR, v=V_CIRC*SPEED_FACTOR, r=URSCRIPT_BLEND)
  movel(apply_correction(p[-0.012858, 0.541260, 0.050005, 3.141576, 0.000000, 0.000000]), a=URSCRIPT_ACCEL*ACCEL_FACTOR, v=V_CIRC*SPEED_FACTOR, r=URSCRIPT_BLEND)
  movel(apply_correction(p[-0.007599, 0.536545, 0.050005, 3.141576, 0.000000, 0.000000]), a=URSCRIPT_ACCEL*ACCEL_FACTOR, v=V_CIRC*SPEED_FACTOR, r=URSCRIPT_BLEND)
  movel(apply_correction(p[-0.001356, 0.539401, 0.050005, 3.141576, 0.000000, 0.000000]), a=URSCRIPT_ACCEL*ACCEL_FACTOR, v=V_CIRC*SPEED_FACTOR, r=URSCRIPT_BLEND)
  movel(apply_correction(p[-0.002041, 0.546340, 0.050005, 3.141576, 0.000000, 0.000000]), a=URSCRIPT_ACCEL*ACCEL_FACTOR, v=V_CIRC*SPEED_FACTOR, r=URSCRIPT_BLEND)
  movel(apply_correction(p[-0.008378, 0.549617, 0.050005, 3.141576, 0.000000, 0.000000]), a=URSCRIPT_ACCEL*ACCEL_FACTOR, v=V_CIRC*SPEED_FACTOR, r=URSCRIPT_BLEND)
  movel(apply_correction(p[-0.015100, 0.547118, 0.050005, 3.141576, 0.000000, 0.000000]), a=URSCRIPT_ACCEL*ACCEL_FACTOR, v=V_CIRC*SPEED_FACTOR, r=URSCRIPT_BLEND)
  movel(apply_correction(p[-0.017677, 0.540470, 0.050005, 3.141576, 0.000000, 0.000000]), a=URSCRIPT_ACCEL*ACCEL_FACTOR, v=V_CIRC*SPEED_FACTOR, r=URSCRIPT_BLEND)
  movel(apply_correction(p[-0.013312, 0.535048, 0.050005, 3.141576, 0.000000, 0.000000]), a=URSCRIPT_ACCEL*ACCEL_FACTOR, v=V_CIRC*SPEED_FACTOR, r=URSCRIPT_BLEND)
  movel(apply_correction(p[-0.006869, 0.537498, 0.050005, 3.141576, 0.000000, 0.000000]), a=URSCRIPT_ACCEL*ACCEL_FACTOR, v=V_CIRC*SPEED_FACTOR, r=URSCRIPT_BLEND)
  movel(apply_correction(p[-0.006196, 0.544557, 0.050005, 3.141576, 0.000000, 0.000000]), a=URSCRIPT_ACCEL*ACCEL_FACTOR, v=V_CIRC*SPEED_FACTOR, r=URSCRIPT_BLEND)
  movel(apply_correction(p[-0.011303, 0.549604, 0.050005, 3.141576, 0.000000, 0.000000]), a=URSCRIPT_ACCEL*ACCEL_FACTOR, v=V_CIRC*SPEED_FACTOR, r=URSCRIPT_BLEND)
  movel(apply_correction(p[-0.018457, 0.549307, 0.050005, 3.141576, 0.000000, 0.000000]), a=URSCRIPT_ACCEL*ACCEL_FACTOR, v=V_CIRC*SPEED_FACTOR, r=URSCRIPT_BLEND)
  movel(apply_correction(p[-0.022436, 0.543491, 0.050005, 3.141576, 0.000000, 0.000000]), a=URSCRIPT_ACCEL*ACCEL_FACTOR, v=V_CIRC*SPEED_FACTOR, r=URSCRIPT_BLEND)
  movel(apply_correction(p[-0.018669, 0.537715, 0.050005, 3.141576, 0.000000, 0.000000]), a=URSCRIPT_ACCEL*ACCEL_FACTOR, v=V_CIRC*SPEED_FACTOR, r=URSCRIPT_BLEND)
  movel(apply_correction(p[-0.011875, 0.539380, 0.050005, 3.141576, 0.000000, 0.000000]), a=URSCRIPT_ACCEL*ACCEL_FACTOR, v=V_CIRC*SPEED_FACTOR, r=URSCRIPT_BLEND)
  movel(apply_correction(p[-0.009742, 0.546188, 0.050005, 3.141576, 0.000000, 0.000000]), a=URSCRIPT_ACCEL*ACCEL_FACTOR, v=V_CIRC*SPEED_FACTOR, r=URSCRIPT_BLEND)
  movel(apply_correction(p[-0.013558, 0.552276, 0.050005, 3.141576, 0.000000, 0.000000]), a=URSCRIPT_ACCEL*ACCEL_FACTOR, v=V_CIRC*SPEED_FACTOR, r=URSCRIPT_BLEND)
  movel(apply_correction(p[-0.020613, 0.553566, 0.050005, 3.141576, 0.000000, 0.000000]), a=URSCRIPT_ACCEL*ACCEL_FACTOR, v=V_CIRC*SPEED_FACTOR, r=URSCRIPT_BLEND)
  movel(apply_correction(p[-0.025840, 0.548787, 0.050005, 3.141576, 0.000000, 0.000000]), a=URSCRIPT_ACCEL*ACCEL_FACTOR, v=V_CIRC*SPEED_FACTOR, r=URSCRIPT_BLEND)
  movel(apply_correction(p[-0.023792, 0.542172, 0.050005, 3.141576, 0.000000, 0.000000]), a=URSCRIPT_ACCEL*ACCEL_FACTOR, v=V_CIRC*SPEED_FACTOR, r=URSCRIPT_BLEND)
  movel(apply_correction(p[-0.016835, 0.542028, 0.050005, 3.141576, 0.000000, 0.000000]), a=URSCRIPT_ACCEL*ACCEL_FACTOR, v=V_CIRC*SPEED_FACTOR, r=URSCRIPT_BLEND)
  movel(apply_correction(p[-0.013339, 0.548221, 0.050005, 3.141576, 0.000000, 0.000000]), a=URSCRIPT_ACCEL*ACCEL_FACTOR, v=V_CIRC*SPEED_FACTOR, r=URSCRIPT_BLEND)
  movel(apply_correction(p[-0.015968, 0.554903, 0.050005, 3.141576, 0.000000, 0.000000]), a=URSCRIPT_ACCEL*ACCEL_FACTOR, v=V_CIRC*SPEED_FACTOR, r=URSCRIPT_BLEND)
  movel(apply_correction(p[-0.022664, 0.557493, 0.050005, 3.141576, 0.000000, 0.000000]), a=URSCRIPT_ACCEL*ACCEL_FACTOR, v=V_CIRC*SPEED_FACTOR, r=URSCRIPT_BLEND)
  movel(apply_correction(p[-0.028833, 0.553959, 0.050005, 3.141576, 0.000000, 0.000000]), a=URSCRIPT_ACCEL*ACCEL_FACTOR, v=V_CIRC*SPEED_FACTOR, r=URSCRIPT_BLEND)
  movel(apply_correction(p[-0.028635, 0.547007, 0.050005, 3.141576, 0.000000, 0.000000]), a=URSCRIPT_ACCEL*ACCEL_FACTOR, v=V_CIRC*SPEED_FACTOR, r=URSCRIPT_BLEND)
  movel(apply_correction(p[-0.022003, 0.545011, 0.050005, 3.141576, 0.000000, 0.000000]), a=URSCRIPT_ACCEL*ACCEL_FACTOR, v=V_CIRC*SPEED_FACTOR, r=URSCRIPT_BLEND)
  movel(apply_correction(p[-0.017259, 0.550270, 0.050005, 3.141576, 0.000000, 0.000000]), a=URSCRIPT_ACCEL*ACCEL_FACTOR, v=V_CIRC*SPEED_FACTOR, r=URSCRIPT_BLEND)
  movel(apply_correction(p[-0.018587, 0.557319, 0.050005, 3.141576, 0.000000, 0.000000]), a=URSCRIPT_ACCEL*ACCEL_FACTOR, v=V_CIRC*SPEED_FACTOR, r=URSCRIPT_BLEND)
  movel(apply_correction(p[-0.024697, 0.561102, 0.050005, 3.141576, 0.000000, 0.000000]), a=URSCRIPT_ACCEL*ACCEL_FACTOR, v=V_CIRC*SPEED_FACTOR, r=URSCRIPT_BLEND)
  movel(apply_correction(p[-0.031491, 0.558927, 0.050005, 3.141576, 0.000000, 0.000000]), a=URSCRIPT_ACCEL*ACCEL_FACTOR, v=V_CIRC*SPEED_FACTOR, r=URSCRIPT_BLEND)
  movel(apply_correction(p[-0.033105, 0.552122, 0.050005, 3.141576, 0.000000, 0.000000]), a=URSCRIPT_ACCEL*ACCEL_FACTOR, v=V_CIRC*SPEED_FACTOR, r=URSCRIPT_BLEND)
  movel(apply_correction(p[-0.027295, 0.548386, 0.050005, 3.141576, 0.000000, 0.000000]), a=URSCRIPT_ACCEL*ACCEL_FACTOR, v=V_CIRC*SPEED_FACTOR, r=URSCRIPT_BLEND)
  movel(apply_correction(p[-0.021500, 0.552402, 0.050005, 3.141576, 0.000000, 0.000000]), a=URSCRIPT_ACCEL*ACCEL_FACTOR, v=V_CIRC*SPEED_FACTOR, r=URSCRIPT_BLEND)
  movel(apply_correction(p[-0.021456, 0.559562, 0.050005, 3.141576, 0.000000, 0.000000]), a=URSCRIPT_ACCEL*ACCEL_FACTOR, v=V_CIRC*SPEED_FACTOR, r=URSCRIPT_BLEND)
  movel(apply_correction(p[-0.026772, 0.564399, 0.050005, 3.141576, 0.000000, 0.000000]), a=URSCRIPT_ACCEL*ACCEL_FACTOR, v=V_CIRC*SPEED_FACTOR, r=URSCRIPT_BLEND)
  movel(apply_correction(p[-0.033883, 0.563631, 0.050005, 3.141576, 0.000000, 0.000000]), a=URSCRIPT_ACCEL*ACCEL_FACTOR, v=V_CIRC*SPEED_FACTOR, r=URSCRIPT_BLEND)
  movel(apply_correction(p[-0.037145, 0.557401, 0.050005, 3.141576, 0.000000, 0.000000]), a=URSCRIPT_ACCEL*ACCEL_FACTOR, v=V_CIRC*SPEED_FACTOR, r=URSCRIPT_BLEND)
  movel(apply_correction(p[-0.032611, 0.552198, 0.050005, 3.141576, 0.000000, 0.000000]), a=URSCRIPT_ACCEL*ACCEL_FACTOR, v=V_CIRC*SPEED_FACTOR, r=URSCRIPT_BLEND)
  movel(apply_correction(p[-0.026054, 0.554687, 0.050005, 3.141576, 0.000000, 0.000000]), a=URSCRIPT_ACCEL*ACCEL_FACTOR, v=V_CIRC*SPEED_FACTOR, r=URSCRIPT_BLEND)
  movel(apply_correction(p[-0.024601, 0.561681, 0.050005, 3.141576, 0.000000, 0.000000]), a=URSCRIPT_ACCEL*ACCEL_FACTOR, v=V_CIRC*SPEED_FACTOR, r=URSCRIPT_BLEND)
  movel(apply_correction(p[-0.028946, 0.567405, 0.050004, 3.141576, 0.000000, 0.000000]), a=URSCRIPT_ACCEL*ACCEL_FACTOR, v=V_CIRC*SPEED_FACTOR, r=URSCRIPT_BLEND)
  movel(apply_correction(p[-0.036085, 0.568036, 0.050004, 3.141576, 0.000000, 0.000000]), a=URSCRIPT_ACCEL*ACCEL_FACTOR, v=V_CIRC*SPEED_FACTOR, r=URSCRIPT_BLEND)
  movel(apply_correction(p[-0.040740, 0.562720, 0.050005, 3.141576, 0.000000, 0.000000]), a=URSCRIPT_ACCEL*ACCEL_FACTOR, v=V_CIRC*SPEED_FACTOR, r=URSCRIPT_BLEND)
  movel(apply_correction(p[-0.037827, 0.556450, 0.050005, 3.141576, 0.000000, 0.000000]), a=URSCRIPT_ACCEL*ACCEL_FACTOR, v=V_CIRC*SPEED_FACTOR, r=URSCRIPT_BLEND)
  movel(apply_correction(p[-0.030891, 0.557198, 0.050005, 3.141576, 0.000000, 0.000000]), a=URSCRIPT_ACCEL*ACCEL_FACTOR, v=V_CIRC*SPEED_FACTOR, r=URSCRIPT_BLEND)
  movel(apply_correction(p[-0.028047, 0.563729, 0.050005, 3.141576, 0.000000, 0.000000]), a=URSCRIPT_ACCEL*ACCEL_FACTOR, v=V_CIRC*SPEED_FACTOR, r=URSCRIPT_BLEND)
  movel(apply_correction(p[-0.031268, 0.570149, 0.050004, 3.141576, 0.000000, 0.000000]), a=URSCRIPT_ACCEL*ACCEL_FACTOR, v=V_CIRC*SPEED_FACTOR, r=URSCRIPT_BLEND)
  movel(apply_correction(p[-0.038167, 0.572121, 0.050004, 3.141576, 0.000000, 0.000000]), a=URSCRIPT_ACCEL*ACCEL_FACTOR, v=V_CIRC*SPEED_FACTOR, r=URSCRIPT_BLEND)
  movel(apply_correction(p[-0.043920, 0.567963, 0.050004, 3.141576, 0.000000, 0.000000]), a=URSCRIPT_ACCEL*ACCEL_FACTOR, v=V_CIRC*SPEED_FACTOR, r=URSCRIPT_BLEND)
  movel(apply_correction(p[-0.042820, 0.561110, 0.050005, 3.141576, 0.000000, 0.000000]), a=URSCRIPT_ACCEL*ACCEL_FACTOR, v=V_CIRC*SPEED_FACTOR, r=URSCRIPT_BLEND)
  end_force_mode()
  movel(apply_correction(p[-0.042820, 0.561110, 0.060005, 3.141576, 0.000000, 0.000000]), a=URSCRIPT_ACCEL*ACCEL_FACTOR, v=0.2500*SPEED_FACTOR)
end

def cycle_4():
  # --- Cycle 4 - Triangulé (0deg) ---
  movel(apply_correction(p[-0.011000, 0.594344, 0.060004, 3.141576, 0.000000, 0.000000]), a=URSCRIPT_ACCEL*ACCEL_FACTOR, v=0.2500*SPEED_FACTOR)
  sleep(0.2)
  zero_ftsensor()
  sleep(0.2)
  force_mode(MEAS_FRAME, [0, 0, 1, 0, 0, 0], [0, 0, -6.0, 0, 0, 0], 2, [0.008, 0.008, 0.04, 0.35, 0.35, 0.35])
  movel(apply_correction(p[-0.011000, 0.594344, 0.045004, 3.141576, 0.000000, 0.000000]), a=URSCRIPT_ACCEL*ACCEL_FACTOR, v=URSCRIPT_RECONTACT_V*SPEED_FACTOR)
  movel(apply_correction(p[-0.011000, 0.594344, 0.050004, 3.141576, 0.000000, 0.000000]), a=URSCRIPT_ACCEL*ACCEL_FACTOR, v=V_RECT*SPEED_FACTOR, r=URSCRIPT_BLEND)
  movel(apply_correction(p[-0.039461, 0.563408, 0.050005, 3.141576, 0.000000, 0.000000]), a=URSCRIPT_ACCEL*ACCEL_FACTOR, v=V_RECT*SPEED_FACTOR, r=URSCRIPT_BLEND)
  movel(apply_correction(p[-0.007288, 0.590632, 0.050004, 3.141576, 0.000000, 0.000000]), a=URSCRIPT_ACCEL*ACCEL_FACTOR, v=V_RECT*SPEED_FACTOR, r=URSCRIPT_BLEND)
  movel(apply_correction(p[-0.034511, 0.558458, 0.050005, 3.141576, 0.000000, 0.000000]), a=URSCRIPT_ACCEL*ACCEL_FACTOR, v=V_RECT*SPEED_FACTOR, r=URSCRIPT_BLEND)
  movel(apply_correction(p[-0.002338, 0.585682, 0.050004, 3.141576, 0.000000, 0.000000]), a=URSCRIPT_ACCEL*ACCEL_FACTOR, v=V_RECT*SPEED_FACTOR, r=URSCRIPT_BLEND)
  movel(apply_correction(p[-0.029562, 0.553509, 0.050005, 3.141576, 0.000000, 0.000000]), a=URSCRIPT_ACCEL*ACCEL_FACTOR, v=V_RECT*SPEED_FACTOR, r=URSCRIPT_BLEND)
  movel(apply_correction(p[0.002612, 0.580732, 0.050004, 3.141576, 0.000000, 0.000000]), a=URSCRIPT_ACCEL*ACCEL_FACTOR, v=V_RECT*SPEED_FACTOR, r=URSCRIPT_BLEND)
  movel(apply_correction(p[-0.024612, 0.548559, 0.050005, 3.141576, 0.000000, 0.000000]), a=URSCRIPT_ACCEL*ACCEL_FACTOR, v=V_RECT*SPEED_FACTOR, r=URSCRIPT_BLEND)
  movel(apply_correction(p[0.007562, 0.575783, 0.050004, 3.141576, 0.000000, 0.000000]), a=URSCRIPT_ACCEL*ACCEL_FACTOR, v=V_RECT*SPEED_FACTOR, r=URSCRIPT_BLEND)
  movel(apply_correction(p[-0.019662, 0.543609, 0.050005, 3.141576, 0.000000, 0.000000]), a=URSCRIPT_ACCEL*ACCEL_FACTOR, v=V_RECT*SPEED_FACTOR, r=URSCRIPT_BLEND)
  movel(apply_correction(p[0.012511, 0.570833, 0.050004, 3.141576, 0.000000, 0.000000]), a=URSCRIPT_ACCEL*ACCEL_FACTOR, v=V_RECT*SPEED_FACTOR, r=URSCRIPT_BLEND)
  movel(apply_correction(p[-0.014712, 0.538659, 0.050005, 3.141576, 0.000000, 0.000000]), a=URSCRIPT_ACCEL*ACCEL_FACTOR, v=V_RECT*SPEED_FACTOR, r=URSCRIPT_BLEND)
  movel(apply_correction(p[0.017461, 0.565883, 0.050004, 3.141576, 0.000000, 0.000000]), a=URSCRIPT_ACCEL*ACCEL_FACTOR, v=V_RECT*SPEED_FACTOR, r=URSCRIPT_BLEND)
  movel(apply_correction(p[-0.011000, 0.534947, 0.050005, 3.141576, 0.000000, 0.000000]), a=URSCRIPT_ACCEL*ACCEL_FACTOR, v=V_RECT*SPEED_FACTOR, r=URSCRIPT_BLEND)
  end_force_mode()
  movel(apply_correction(p[-0.011000, 0.534947, 0.060005, 3.141576, 0.000000, 0.000000]), a=URSCRIPT_ACCEL*ACCEL_FACTOR, v=0.2500*SPEED_FACTOR)
end

def cycle_5():
  # --- Cycle 5 - Triangulé (90deg) ---
  movel(apply_correction(p[-0.040698, 0.564646, 0.060005, 3.141576, 0.000000, 0.000000]), a=URSCRIPT_ACCEL*ACCEL_FACTOR, v=0.2500*SPEED_FACTOR)
  sleep(0.2)
  zero_ftsensor()
  sleep(0.2)
  force_mode(MEAS_FRAME, [0, 0, 1, 0, 0, 0], [0, 0, -6.0, 0, 0, 0], 2, [0.008, 0.008, 0.04, 0.35, 0.35, 0.35])
  movel(apply_correction(p[-0.040698, 0.564646, 0.045005, 3.141576, 0.000000, 0.000000]), a=URSCRIPT_ACCEL*ACCEL_FACTOR, v=URSCRIPT_RECONTACT_V*SPEED_FACTOR)
  movel(apply_correction(p[-0.040698, 0.564646, 0.050005, 3.141576, 0.000000, 0.000000]), a=URSCRIPT_ACCEL*ACCEL_FACTOR, v=V_RECT*SPEED_FACTOR, r=URSCRIPT_BLEND)
  movel(apply_correction(p[-0.009763, 0.536185, 0.050005, 3.141576, 0.000000, 0.000000]), a=URSCRIPT_ACCEL*ACCEL_FACTOR, v=V_RECT*SPEED_FACTOR, r=URSCRIPT_BLEND)
  movel(apply_correction(p[-0.036986, 0.568358, 0.050004, 3.141576, 0.000000, 0.000000]), a=URSCRIPT_ACCEL*ACCEL_FACTOR, v=V_RECT*SPEED_FACTOR, r=URSCRIPT_BLEND)
  movel(apply_correction(p[-0.004813, 0.541134, 0.050005, 3.141576, 0.000000, 0.000000]), a=URSCRIPT_ACCEL*ACCEL_FACTOR, v=V_RECT*SPEED_FACTOR, r=URSCRIPT_BLEND)
  movel(apply_correction(p[-0.032036, 0.573308, 0.050004, 3.141576, 0.000000, 0.000000]), a=URSCRIPT_ACCEL*ACCEL_FACTOR, v=V_RECT*SPEED_FACTOR, r=URSCRIPT_BLEND)
  movel(apply_correction(p[0.000137, 0.546084, 0.050005, 3.141576, 0.000000, 0.000000]), a=URSCRIPT_ACCEL*ACCEL_FACTOR, v=V_RECT*SPEED_FACTOR, r=URSCRIPT_BLEND)
  movel(apply_correction(p[-0.027087, 0.578257, 0.050004, 3.141576, 0.000000, 0.000000]), a=URSCRIPT_ACCEL*ACCEL_FACTOR, v=V_RECT*SPEED_FACTOR, r=URSCRIPT_BLEND)
  movel(apply_correction(p[0.005087, 0.551034, 0.050005, 3.141576, 0.000000, 0.000000]), a=URSCRIPT_ACCEL*ACCEL_FACTOR, v=V_RECT*SPEED_FACTOR, r=URSCRIPT_BLEND)
  movel(apply_correction(p[-0.022137, 0.583207, 0.050004, 3.141576, 0.000000, 0.000000]), a=URSCRIPT_ACCEL*ACCEL_FACTOR, v=V_RECT*SPEED_FACTOR, r=URSCRIPT_BLEND)
  movel(apply_correction(p[0.010036, 0.555984, 0.050005, 3.141576, 0.000000, 0.000000]), a=URSCRIPT_ACCEL*ACCEL_FACTOR, v=V_RECT*SPEED_FACTOR, r=URSCRIPT_BLEND)
  movel(apply_correction(p[-0.017187, 0.588157, 0.050004, 3.141576, 0.000000, 0.000000]), a=URSCRIPT_ACCEL*ACCEL_FACTOR, v=V_RECT*SPEED_FACTOR, r=URSCRIPT_BLEND)
  movel(apply_correction(p[0.014986, 0.560933, 0.050005, 3.141576, 0.000000, 0.000000]), a=URSCRIPT_ACCEL*ACCEL_FACTOR, v=V_RECT*SPEED_FACTOR, r=URSCRIPT_BLEND)
  movel(apply_correction(p[-0.012237, 0.593107, 0.050004, 3.141576, 0.000000, 0.000000]), a=URSCRIPT_ACCEL*ACCEL_FACTOR, v=V_RECT*SPEED_FACTOR, r=URSCRIPT_BLEND)
  movel(apply_correction(p[0.018698, 0.564646, 0.050005, 3.141576, 0.000000, 0.000000]), a=URSCRIPT_ACCEL*ACCEL_FACTOR, v=V_RECT*SPEED_FACTOR, r=URSCRIPT_BLEND)
  end_force_mode()
  movel(apply_correction(p[0.018698, 0.564646, 0.060005, 3.141576, 0.000000, 0.000000]), a=URSCRIPT_ACCEL*ACCEL_FACTOR, v=0.2500*SPEED_FACTOR)
end

def cycle_6():
  # --- Cycle 6 - Triangulé (0deg) ---
  movel(apply_correction(p[-0.011000, 0.594344, 0.060004, 3.141576, 0.000000, 0.000000]), a=URSCRIPT_ACCEL*ACCEL_FACTOR, v=0.2500*SPEED_FACTOR)
  sleep(0.2)
  zero_ftsensor()
  sleep(0.2)
  force_mode(MEAS_FRAME, [0, 0, 1, 0, 0, 0], [0, 0, -6.0, 0, 0, 0], 2, [0.008, 0.008, 0.04, 0.35, 0.35, 0.35])
  movel(apply_correction(p[-0.011000, 0.594344, 0.045004, 3.141576, 0.000000, 0.000000]), a=URSCRIPT_ACCEL*ACCEL_FACTOR, v=URSCRIPT_RECONTACT_V*SPEED_FACTOR)
  movel(apply_correction(p[-0.011000, 0.594344, 0.050004, 3.141576, 0.000000, 0.000000]), a=URSCRIPT_ACCEL*ACCEL_FACTOR, v=V_RECT*SPEED_FACTOR, r=URSCRIPT_BLEND)
  movel(apply_correction(p[-0.039461, 0.563408, 0.050005, 3.141576, 0.000000, 0.000000]), a=URSCRIPT_ACCEL*ACCEL_FACTOR, v=V_RECT*SPEED_FACTOR, r=URSCRIPT_BLEND)
  movel(apply_correction(p[-0.007288, 0.590632, 0.050004, 3.141576, 0.000000, 0.000000]), a=URSCRIPT_ACCEL*ACCEL_FACTOR, v=V_RECT*SPEED_FACTOR, r=URSCRIPT_BLEND)
  movel(apply_correction(p[-0.034511, 0.558458, 0.050005, 3.141576, 0.000000, 0.000000]), a=URSCRIPT_ACCEL*ACCEL_FACTOR, v=V_RECT*SPEED_FACTOR, r=URSCRIPT_BLEND)
  movel(apply_correction(p[-0.002338, 0.585682, 0.050004, 3.141576, 0.000000, 0.000000]), a=URSCRIPT_ACCEL*ACCEL_FACTOR, v=V_RECT*SPEED_FACTOR, r=URSCRIPT_BLEND)
  movel(apply_correction(p[-0.029562, 0.553509, 0.050005, 3.141576, 0.000000, 0.000000]), a=URSCRIPT_ACCEL*ACCEL_FACTOR, v=V_RECT*SPEED_FACTOR, r=URSCRIPT_BLEND)
  movel(apply_correction(p[0.002612, 0.580732, 0.050004, 3.141576, 0.000000, 0.000000]), a=URSCRIPT_ACCEL*ACCEL_FACTOR, v=V_RECT*SPEED_FACTOR, r=URSCRIPT_BLEND)
  movel(apply_correction(p[-0.024612, 0.548559, 0.050005, 3.141576, 0.000000, 0.000000]), a=URSCRIPT_ACCEL*ACCEL_FACTOR, v=V_RECT*SPEED_FACTOR, r=URSCRIPT_BLEND)
  movel(apply_correction(p[0.007562, 0.575783, 0.050004, 3.141576, 0.000000, 0.000000]), a=URSCRIPT_ACCEL*ACCEL_FACTOR, v=V_RECT*SPEED_FACTOR, r=URSCRIPT_BLEND)
  movel(apply_correction(p[-0.019662, 0.543609, 0.050005, 3.141576, 0.000000, 0.000000]), a=URSCRIPT_ACCEL*ACCEL_FACTOR, v=V_RECT*SPEED_FACTOR, r=URSCRIPT_BLEND)
  movel(apply_correction(p[0.012511, 0.570833, 0.050004, 3.141576, 0.000000, 0.000000]), a=URSCRIPT_ACCEL*ACCEL_FACTOR, v=V_RECT*SPEED_FACTOR, r=URSCRIPT_BLEND)
  movel(apply_correction(p[-0.014712, 0.538659, 0.050005, 3.141576, 0.000000, 0.000000]), a=URSCRIPT_ACCEL*ACCEL_FACTOR, v=V_RECT*SPEED_FACTOR, r=URSCRIPT_BLEND)
  movel(apply_correction(p[0.017461, 0.565883, 0.050004, 3.141576, 0.000000, 0.000000]), a=URSCRIPT_ACCEL*ACCEL_FACTOR, v=V_RECT*SPEED_FACTOR, r=URSCRIPT_BLEND)
  movel(apply_correction(p[-0.011000, 0.534947, 0.050005, 3.141576, 0.000000, 0.000000]), a=URSCRIPT_ACCEL*ACCEL_FACTOR, v=V_RECT*SPEED_FACTOR, r=URSCRIPT_BLEND)
  end_force_mode()
  movel(apply_correction(p[-0.011000, 0.534947, 0.060005, 3.141576, 0.000000, 0.000000]), a=URSCRIPT_ACCEL*ACCEL_FACTOR, v=0.2500*SPEED_FACTOR)
end

def etalement():
  set_tcp(p[0.0, 0.0, 0.2657, 0, 0, 0])
  # Aucune pose home absolue : la position de depart est la pose courante
  # du robot (mesuree a l'execution). L'operateur jogge le robot ou il
  # veut, clique Start, et le sondage de surface part de la.
  home = get_actual_tcp_pose()
  probe_surface_z()

  cycle_1()
  cycle_2()
  cycle_3()
  cycle_4()
  cycle_5()
  cycle_6()
  movel(apply_correction(p[-0.011000, 0.534947, 0.080005, 3.141576, 0.000000, 0.000000]), a=URSCRIPT_ACCEL*ACCEL_FACTOR, v=0.2500*SPEED_FACTOR)
end

etalement()
